Omron CX-Programmer project NewProject (CX-Programmer 9.73)

# PLC NodeA: CP2E-N N

## Global symbols (name address type ; comment)
0 CHANNEL  ; Value
0.00 BOOL  ; MSET
0.01 BOOL  ; AUTO
0.02 BOOL  ; ALRM
0.03 BOOL  ; QMC
0.04 BOOL  ; STRB
0.05 BOOL  ; CNTR
0.06 BOOL  ; 1
0.07 BOOL  ; 2
0.08 BOOL  ; 4
0.09 BOOL  ; 8
0.10 BOOL  ; 16
0.11 BOOL  ; 32
1 CHANNEL  ; Value
D10000 CHANNEL  ; MSET
D10001 CHANNEL  ; AUTO
D10002 CHANNEL  ; ALRM
D10003 CHANNEL  ; QMC
D10004 CHANNEL  ; STRB
D10005 CHANNEL  ; CNTR
D10006 CHANNEL  ; 1
D10007 CHANNEL  ; 2
D10008 CHANNEL  ; 4
D10009 CHANNEL  ; 8
D10010 CHANNEL  ; 16
D10011 CHANNEL  ; 32
D9000 CHANNEL  ; Node_ErrorCode
D9001 CHANNEL  ; NodeC_Errorcode
D9002 CHANNEL  ; NodeD_ErrorCode
W10.00 BOOL  ; Node_link
W10.01 BOOL  ; Node_BUSY
W10.02 BOOL  ; Node_OK
W10.03 BOOL  ; Node_NG
W11.00 BOOL  ; NodeC_link
W11.01 BOOL  ; NodeC_BUSY
W11.02 BOOL  ; NodeC_OK
W11.03 BOOL  ; NodeC_NG
W12.00 BOOL  ; NodeD_link
W12.01 BOOL  ; NodeD_BUSY
W12.02 BOOL  ; NodeD_OK
W12.03 BOOL  ; NodeD_NG
FINS_DCS _CPxx001_SendData
FINS_Ethernet _CPxx001_SendData
Send_NodeB _CPxx001_SendData
Send_NodeC _CPxx001_SendData
Send_NodeD _CPxx001_SendData

## Program NewProgram1 (cyclic task 0)

### Section Section1

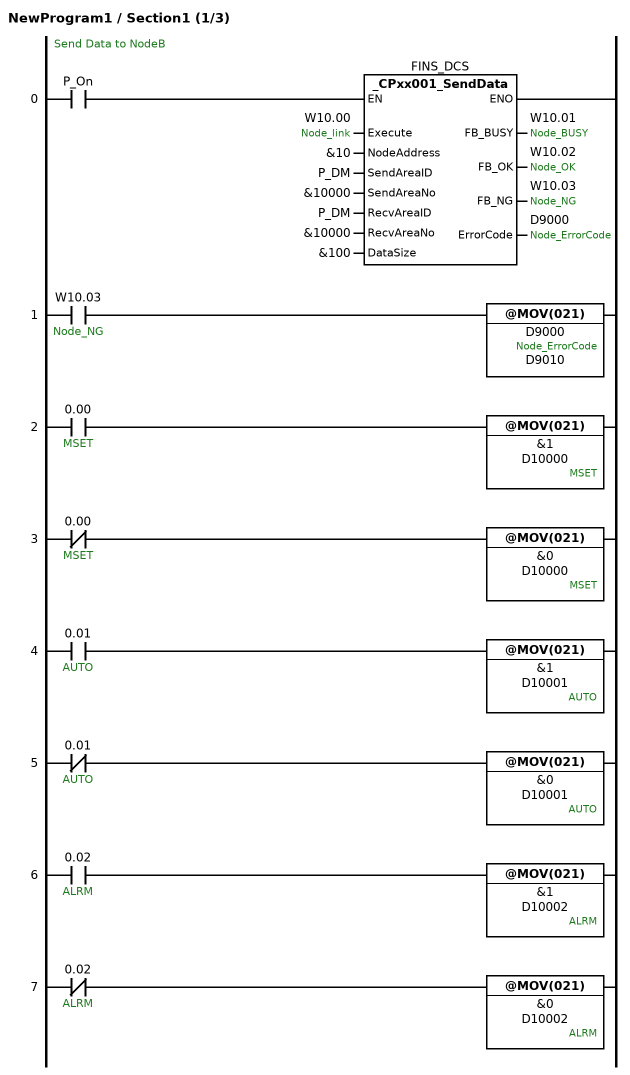
; rung 0: Send Data to NodeB
LD P_On
CALL FINS_DCS : _CPxx001_SendData (Execute := W10.00, NodeAddress := &10, SendAreaID := P_DM, SendAreaNo := &10000, RecvAreaID := P_DM, RecvAreaNo := &10000, DataSize := &100, FB_BUSY => W10.01, FB_OK => W10.02, FB_NG => W10.03, ErrorCode => D9000)  ; Node_link, Node_BUSY, Node_OK, Node_NG, Node_ErrorCode
; rung 1
LD W10.03  ; Node_NG
@MOV(021) D9000 D9010  ; Node_ErrorCode
; rung 2
LD 0.00  ; MSET
@MOV(021) &1 D10000  ; MSET
; rung 3
LDNOT 0.00  ; MSET
@MOV(021) &0 D10000  ; MSET
; rung 4
LD 0.01  ; AUTO
@MOV(021) &1 D10001  ; AUTO
; rung 5
LDNOT 0.01  ; AUTO
@MOV(021) &0 D10001  ; AUTO
; rung 6
LD 0.02  ; ALRM
@MOV(021) &1 D10002  ; ALRM
; rung 7
LDNOT 0.02  ; ALRM
@MOV(021) &0 D10002  ; ALRM

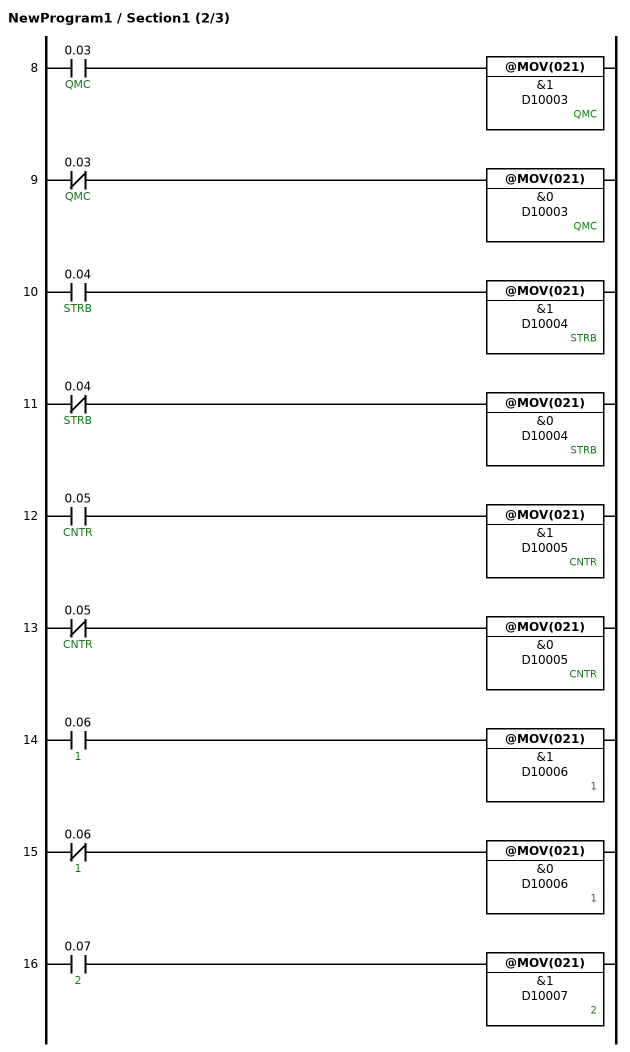
; rung 8
LD 0.03  ; QMC
@MOV(021) &1 D10003  ; QMC
; rung 9
LDNOT 0.03  ; QMC
@MOV(021) &0 D10003  ; QMC
; rung 10
LD 0.04  ; STRB
@MOV(021) &1 D10004  ; STRB
; rung 11
LDNOT 0.04  ; STRB
@MOV(021) &0 D10004  ; STRB
; rung 12
LD 0.05  ; CNTR
@MOV(021) &1 D10005  ; CNTR
; rung 13
LDNOT 0.05  ; CNTR
@MOV(021) &0 D10005  ; CNTR
; rung 14
LD 0.06  ; 1
@MOV(021) &1 D10006  ; 1
; rung 15
LDNOT 0.06  ; 1
@MOV(021) &0 D10006  ; 1
; rung 16
LD 0.07  ; 2
@MOV(021) &1 D10007  ; 2

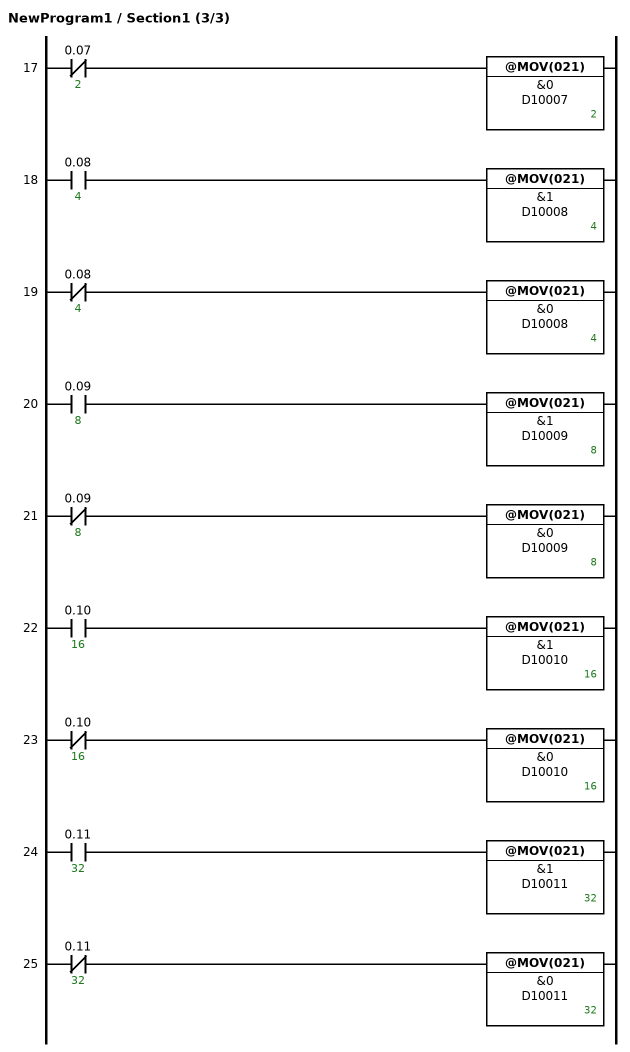
; rung 17
LDNOT 0.07  ; 2
@MOV(021) &0 D10007  ; 2
; rung 18
LD 0.08  ; 4
@MOV(021) &1 D10008  ; 4
; rung 19
LDNOT 0.08  ; 4
@MOV(021) &0 D10008  ; 4
; rung 20
LD 0.09  ; 8
@MOV(021) &1 D10009  ; 8
; rung 21
LDNOT 0.09  ; 8
@MOV(021) &0 D10009  ; 8
; rung 22
LD 0.10  ; 16
@MOV(021) &1 D10010  ; 16
; rung 23
LDNOT 0.10  ; 16
@MOV(021) &0 D10010  ; 16
; rung 24
LD 0.11  ; 32
@MOV(021) &1 D10011  ; 32
; rung 25
LDNOT 0.11  ; 32
@MOV(021) &0 D10011  ; 32

### Section END
; rung 0
END(001)

## Function block _CPxx001_SendData (Omron library block, body left out)